Staubli VAL3: getDetectFrame.pgx

public program getDetectFrame(frame& x_fDetection, frame x_fRefFrame, num& x_nError)
  local string l_sCustomTxt[2]
begin
  // This program returns the position of the conveyor frame
  // in the réference frame passed as parameter
  //
  // Input param
  //  x_fRefFrame   : Reference frame in which the position of the conveyor
  //                frame must be returned
  //
  // Output param
  //  x_fConveyor   : Conveyor frame
  //  x_nError      : Error code
  //    0    --> No error
  //    14   --> Conveyor library not started, the frame cannot be computed.
  //
  // Created 7-03-08                                   C.CURRIVAND
  //----------------------------------------------------------------
  x_nError=0
  if bInit
    x_fDetection.trsf=position(fDetection,x_fRefFrame)
  else
    x_nError=14
    // Prepare clear text error message
    l_sCustomTxt[0]=sConveyorName
    l_sCustomTxt[1]="detection"
    call ut:addStrToString(lang:sListOfMessage[x_nError],sErrorMessage,"",l_sCustomTxt)
  endIf
end
